TYPE ID50FIFOBuffer :
STRUCT
	Size: UDINT := 50;
	Buffer: ARRAY [0..49] OF ComponentIdentifier;
END_STRUCT
END_TYPE

(* stored: Version 1.1.0.1, ProductVersion 3.1.4024.9
   DUT ID50FIFOBuffer: Id {354de428-b430-4693-a55e-3f71e7611f95} *)
